FUNCTION_BLOCK ASSEMBLE_AB_FROM_AX (* this Function combines the 8 AX (BOOL) adapters to a AB (BYTE) *)
  (* Standard: 61499-2; Description: Copyright (c) 2025 Meisterschulen am Ostbahnhof This program and the accompanying materials are made available under the terms of the Eclipse Public License 2.0 which is available at https://www.eclipse.org/legal/epl-2.0/ SPDX-License-Identifier: EPL-2.0 *)
  (* Version 1.0, 2026-03-05, Franz Höpfinger, Meisterschulen am Ostbahnhof, initial API and implementation and/or initial documentation *)
  PACKAGE adapter::assembling;
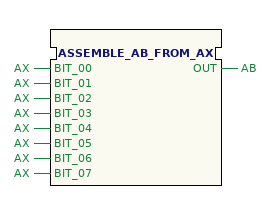
  SOCKETS
    BIT_00 : adapter::types::unidirectional::AX; (* Bool Bit 0 *)
    BIT_01 : adapter::types::unidirectional::AX; (* Bool Bit 1 *)
    BIT_02 : adapter::types::unidirectional::AX; (* Bool Bit 2 *)
    BIT_03 : adapter::types::unidirectional::AX; (* Bool Bit 3 *)
    BIT_04 : adapter::types::unidirectional::AX; (* Bool Bit 4 *)
    BIT_05 : adapter::types::unidirectional::AX; (* Bool Bit 5 *)
    BIT_06 : adapter::types::unidirectional::AX; (* Bool Bit 6 *)
    BIT_07 : adapter::types::unidirectional::AX; (* Bool Bit 7 *)
  END_SOCKETS
  PLUGS
    OUT : adapter::types::unidirectional::AB; (* BYTE Output *)
  END_PLUGS
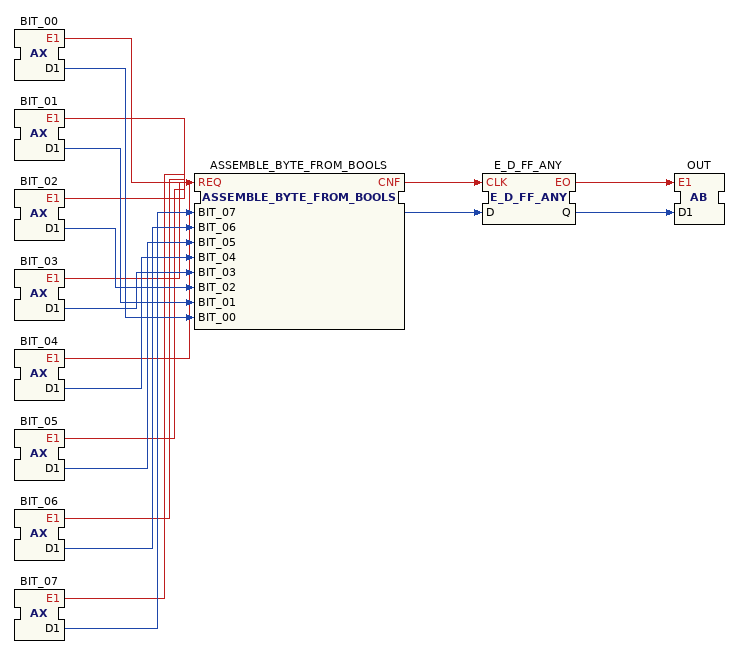
  FBS
    ASSEMBLE_BYTE_FROM_BOOLS : eclipse4diac::utils::assembling::ASSEMBLE_BYTE_FROM_BOOLS;
    E_D_FF_ANY : iec61499::events::E_D_FF_ANY;
  END_FBS
  EVENT_CONNECTIONS
    BIT_00.E1 TO ASSEMBLE_BYTE_FROM_BOOLS.REQ;
    BIT_01.E1 TO ASSEMBLE_BYTE_FROM_BOOLS.REQ;
    BIT_02.E1 TO ASSEMBLE_BYTE_FROM_BOOLS.REQ;
    BIT_03.E1 TO ASSEMBLE_BYTE_FROM_BOOLS.REQ;
    BIT_04.E1 TO ASSEMBLE_BYTE_FROM_BOOLS.REQ;
    BIT_05.E1 TO ASSEMBLE_BYTE_FROM_BOOLS.REQ;
    BIT_06.E1 TO ASSEMBLE_BYTE_FROM_BOOLS.REQ;
    BIT_07.E1 TO ASSEMBLE_BYTE_FROM_BOOLS.REQ;
    ASSEMBLE_BYTE_FROM_BOOLS.CNF TO E_D_FF_ANY.CLK;
    E_D_FF_ANY.EO TO OUT.E1;
  END_CONNECTIONS
  DATA_CONNECTIONS
    ASSEMBLE_BYTE_FROM_BOOLS. TO E_D_FF_ANY.D;
    E_D_FF_ANY.Q TO OUT.D1;
    BIT_07.D1 TO ASSEMBLE_BYTE_FROM_BOOLS.BIT_07;
    BIT_06.D1 TO ASSEMBLE_BYTE_FROM_BOOLS.BIT_06;
    BIT_05.D1 TO ASSEMBLE_BYTE_FROM_BOOLS.BIT_05;
    BIT_04.D1 TO ASSEMBLE_BYTE_FROM_BOOLS.BIT_04;
    BIT_03.D1 TO ASSEMBLE_BYTE_FROM_BOOLS.BIT_03;
    BIT_02.D1 TO ASSEMBLE_BYTE_FROM_BOOLS.BIT_02;
    BIT_01.D1 TO ASSEMBLE_BYTE_FROM_BOOLS.BIT_01;
    BIT_00.D1 TO ASSEMBLE_BYTE_FROM_BOOLS.BIT_00;
  END_CONNECTIONS
END_FUNCTION_BLOCK
